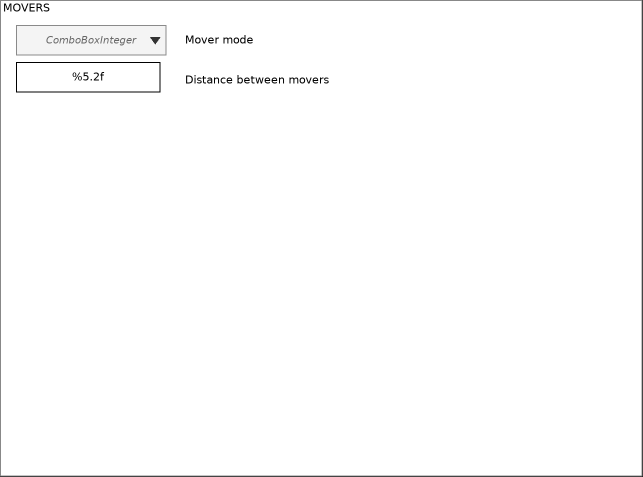
VISUALIZATION VI_XTSMoversConfigurationVisu  // 643x477
VAR_IN_OUT
	xts : XTS_System;
END_VAR
VAR
	stTableStruct : ARRAY [1..25] OF stTableStructx10;
END_VAR
    Rectangle (0,0 643x477), "MOVERS"
    Label (182,25 150x30), "Mover mode"
    ComboBoxInteger (16,25 150x30), variable: xts.stCfg.udiMoverMode, text list: 'MoverMode_TXT'
    Label (182,65 150x30), "Distance between movers"
    Rectangle (16,62 144x30), "%5.2f", text variable: xts.stCfg.lrMoverDistance
        OnMouseClick: write the text variable via Default
END_VISUALIZATION

(* stored: Version 1.1.0.1, ProductVersion 3.1.4024.11
   Visu VI_XTSMoversConfigurationVisu: Id {91fbc901-a7c8-4f77-a3e0-550592c41db5} *)
